KUKA KRL program: ab_com_01_st01_g01.src, ab_com_01_st01_g01.dat

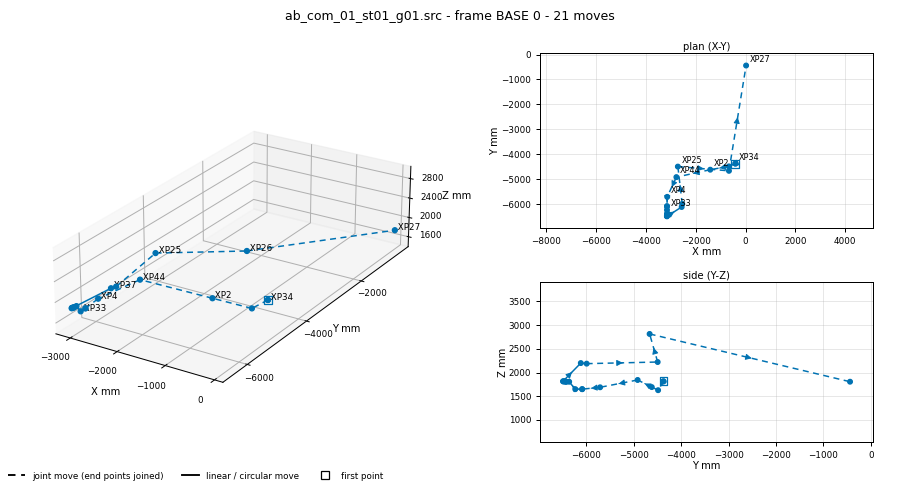
[picture p0: tool path of ab_com_01_st01_g01.src in frame BASE 0, 21 of 21 moves have a stored position in this frame; points joined in program order, loops and branches not executed]
--- ab_com_01_st01_g01.src ---
&ACCESS RVP1
&REL 2213
&COMMENT Deposito Frente AXOR_ATEGO
&PARAM DISKPATH = KRC:\R1\Program\OLP
&PARAM TEMPLATE = C:\KRC\Roboter\Template\vorgabe
&PARAM EDITMASK = *
DEF AB_COM_01_ST01_G01( )
;FOLD INI
  ;FOLD BASISTECH INI
    GLOBAL INTERRUPT DECL 3 WHEN $STOPMESS==TRUE DO IR_STOPM ( )
    INTERRUPT ON 3
    BAS (#INITMOV,0 )
  ;ENDFOLD (BASISTECH INI)
;FOLD SPOTTECH INI
USERSPOT(#INIT)
;ENDFOLD (SPOTTECH INI)
;FOLD GRIPPERTECH INI
USER_GRP(0,DUMMY,DUMMY,GDEFAULT)
;ENDFOLD (GRIPPERTECH INI)
  ;FOLD USER INI
    ;Make your modifications here

  ;ENDFOLD (USER INI)
;ENDFOLD (INI)

; Caracterização dos meios de produção
; Changes: Deposita Frontal na GeoBox
; Modelos:Atego/Axor - ETB/LTA/LTB/STB
; Versão Atual:28/03/2016
; Name: P13.050-R4

chk_w6_wechs_ok ( )  ; CHECK GRIPPER AXOR/ATEGO

;FOLD PTP P34 CONT Vel=100 % PDAT16 Tool[7]:Gripper Geo G01 01 Base[0] CD;%{PE}%R 8.2.20,%MKUKATPBASIS,%CMOVE,%VPTP,%P 1:PTP, 2:P34, 3:C_DIS, 5:100, 7:PDAT16
$BWDSTART=FALSE
PDAT_ACT=PPDAT16
FDAT_ACT=FP34
BAS(#PTP_PARAMS,100)
PTP XP34 C_DIS
;ENDFOLD

;FOLD PTP P7 Vel=100 % PDAT6 Tool[7]:Gripper Geo G01 01 Base[0];%{PE}%R 8.2.20,%MKUKATPBASIS,%CMOVE,%VPTP,%P 1:PTP, 2:P7, 3:, 5:100, 7:PDAT6
$BWDSTART=FALSE
PDAT_ACT=PPDAT6
FDAT_ACT=FP7
BAS(#PTP_PARAMS,100)
PTP XP7
;ENDFOLD

;FOLD OUT 3372 'Lib. pré Dep. Axor/Atego' State=TRUE ;%{PE}%R 8.2.20,%MKUKATPBASIS,%COUT,%VOUTX,%P 2:3372, 3:Lib. pré Dep. Axor/Atego, 5:TRUE, 6:
$OUT[3372]=TRUE
;ENDFOLD
;FOLD WAIT FOR ( IN 3372 'Lib. pré Deposito Axor/Atego' );%{PE}%R 8.2.20,%MKUKATPBASIS,%CEXT_WAIT_FOR,%VEXT_WAIT_FOR,%P 2:, 4:, 5:$IN, 6:3372, 7:Lib. pré Deposito Axor/Atego, 9:
WAIT FOR  ( $IN[3372] )
;ENDFOLD
;FOLD OUT 3372 'Lib. pré Dep. Axor/Atego' State=FALSE ;%{PE}%R 8.2.20,%MKUKATPBASIS,%COUT,%VOUTX,%P 2:3372, 3:Lib. pré Dep. Axor/Atego, 5:FALSE, 6:
$OUT[3372]=FALSE
;ENDFOLD
;FOLD OUT 3348 'Fora area GEOBOX' State=FALSE ;%{PE}%R 8.2.20,%MKUKATPBASIS,%COUT,%VOUTX,%P 2:3348, 3:Fora area GEOBOX, 5:FALSE, 6:
$OUT[3348]=FALSE
;ENDFOLD
;FOLD OUT 3340 'Area_Clear_AGV' State=FALSE ;%{PE}%R 8.2.20,%MKUKATPBASIS,%COUT,%VOUTX,%P 2:3340, 3:Area_Clear_AGV, 5:FALSE, 6:
$OUT[3340]=FALSE
;ENDFOLD

;FOLD PTP P1 CONT Vel=100 % PDAT1 Tool[7]:Gripper Geo G01 01 Base[0] CD;%{PE}%R 8.2.20,%MKUKATPBASIS,%CMOVE,%VPTP,%P 1:PTP, 2:P1, 3:C_DIS, 5:100, 7:PDAT1
$BWDSTART=FALSE
PDAT_ACT=PPDAT1
FDAT_ACT=FP1
BAS(#PTP_PARAMS,100)
PTP XP1 C_DIS
;ENDFOLD
;FOLD PTP P2 CONT Vel=100 % PDAT2 Tool[7]:Gripper Geo G01 01 Base[0] CD;%{PE}%R 8.2.20,%MKUKATPBASIS,%CMOVE,%VPTP,%P 1:PTP, 2:P2, 3:C_DIS, 5:100, 7:PDAT2
$BWDSTART=FALSE
PDAT_ACT=PPDAT2
FDAT_ACT=FP2
BAS(#PTP_PARAMS,100)
PTP XP2 C_DIS
;ENDFOLD
;FOLD PTP P44 CONT Vel=100 % PDAT27 Tool[7]:Gripper Geo G01 01 Base[0];%{PE}%R 8.2.20,%MKUKATPBASIS,%CMOVE,%VPTP,%P 1:PTP, 2:P44, 3:C_DIS, 5:100, 7:PDAT27
$BWDSTART=FALSE
PDAT_ACT=PPDAT27
FDAT_ACT=FP44
BAS(#PTP_PARAMS,100)
PTP XP44 C_DIS
;ENDFOLD
;FOLD PTP P4 CONT Vel=100 % PDAT8 Tool[7]:Gripper Geo G01 01 Base[0] CD;%{PE}%R 8.2.20,%MKUKATPBASIS,%CMOVE,%VPTP,%P 1:PTP, 2:P4, 3:C_DIS, 5:100, 7:PDAT8
$BWDSTART=FALSE
PDAT_ACT=PPDAT8
FDAT_ACT=FP4
BAS(#PTP_PARAMS,100)
PTP XP4 C_DIS
;ENDFOLD

;FOLD ; ABRE GRAMPOS E VERIFICA;%{PE}%R 8.2.20,%MKUKATPBASIS,%CCOMMENT,%VNORMAL,%P 2:ABRE  GRAMPOS  E  VERIFICA
;ENDFOLD
;FOLD SET Z3.1/Z3.2 AXOR State= GDAT20;%{PE}%R 8.2.1,%MKUKATPGRP,%CGRP,%VGRP,%P 2:7, 4:1, 5:#NO, 6:GDAT20, 8:0, 10:0
H50(GRP,7,1,GGDAT20)
;ENDFOLD
chk_w6_grp3_opn ()

;FOLD OUT 3374 'Lib. Dep. Axor/Atego' State=TRUE ;%{PE}%R 8.2.20,%MKUKATPBASIS,%COUT,%VOUTX,%P 2:3374, 3:Lib. Dep. Axor/Atego, 5:TRUE, 6:
$OUT[3374]=TRUE
;ENDFOLD
;FOLD WAIT FOR ( IN 3374 'Lib. Deposito Axor/Atego' );%{PE}%R 8.2.20,%MKUKATPBASIS,%CEXT_WAIT_FOR,%VEXT_WAIT_FOR,%P 2:, 4:, 5:$IN, 6:3374, 7:Lib. Deposito Axor/Atego, 9:
WAIT FOR  ( $IN[3374] )
;ENDFOLD
;FOLD OUT 3374 'Lib. Dep. Axor/Atego' State=FALSE ;%{PE}%R 8.2.20,%MKUKATPBASIS,%COUT,%VOUTX,%P 2:3374, 3:Lib. Dep. Axor/Atego, 5:FALSE, 6:
$OUT[3374]=FALSE
;ENDFOLD

;FOLD PTP P9 Vel=100 % PDAT11 Tool[7]:Gripper Geo G01 01 Base[0];%{PE}%R 8.2.20,%MKUKATPBASIS,%CMOVE,%VPTP,%P 1:PTP, 2:P9, 3:, 5:100, 7:PDAT11
$BWDSTART=FALSE
PDAT_ACT=PPDAT11
FDAT_ACT=FP9
BAS(#PTP_PARAMS,100)
PTP XP9
;ENDFOLD
;FOLD LIN P32 CONT Vel=0.5 m/s CPDAT20 Tool[7]:Gripper Geo G01 01 Base[0] CD;%{PE}%R 8.2.20,%MKUKATPBASIS,%CMOVE,%VLIN,%P 1:LIN, 2:P32, 3:C_DIS C_DIS, 5:0.5, 7:CPDAT20
$BWDSTART=FALSE
LDAT_ACT=LCPDAT20
FDAT_ACT=FP32
BAS(#CP_PARAMS,0.5)
LIN XP32 C_DIS C_DIS
;ENDFOLD
;FOLD LIN P33 CONT Vel=0.5 m/s CPDAT21 Tool[7]:Gripper Geo G01 01 Base[0] CD;%{PE}%R 8.2.20,%MKUKATPBASIS,%CMOVE,%VLIN,%P 1:LIN, 2:P33, 3:C_DIS C_DIS, 5:0.5, 7:CPDAT21
$BWDSTART=FALSE
LDAT_ACT=LCPDAT21
FDAT_ACT=FP33
BAS(#CP_PARAMS,0.5)
LIN XP33 C_DIS C_DIS
;ENDFOLD
;FOLD LIN P10 CONT Vel=0.5 m/s CPDAT4 Tool[7]:Gripper Geo G01 01 Base[0] CD;%{PE}%R 8.2.20,%MKUKATPBASIS,%CMOVE,%VLIN,%P 1:LIN, 2:P10, 3:C_DIS C_DIS, 5:0.5, 7:CPDAT4
$BWDSTART=FALSE
LDAT_ACT=LCPDAT4
FDAT_ACT=FP10
BAS(#CP_PARAMS,0.5)
LIN XP10 C_DIS C_DIS
;ENDFOLD
;FOLD LIN P5 CONT Vel=0.5 m/s CPDAT8 Tool[7]:Gripper Geo G01 01 Base[0] CD;%{PE}%R 8.2.20,%MKUKATPBASIS,%CMOVE,%VLIN,%P 1:LIN, 2:P5, 3:C_DIS C_DIS, 5:0.5, 7:CPDAT8
$BWDSTART=FALSE
LDAT_ACT=LCPDAT8
FDAT_ACT=FP5
BAS(#CP_PARAMS,0.5)
LIN XP5 C_DIS C_DIS
;ENDFOLD
;FOLD LIN P36 CONT Vel=0.5 m/s CPDAT22 Tool[7]:Gripper Geo G01 01 Base[0] CD;%{PE}%R 8.2.20,%MKUKATPBASIS,%CMOVE,%VLIN,%P 1:LIN, 2:P36, 3:C_DIS C_DIS, 5:0.5, 7:CPDAT22
$BWDSTART=FALSE
LDAT_ACT=LCPDAT22
FDAT_ACT=FP36
BAS(#CP_PARAMS,0.5)
LIN XP36 C_DIS C_DIS
;ENDFOLD
;FOLD LIN P17 CONT Vel=0.5 m/s CPDAT12 Tool[7]:Gripper Geo G01 01 Base[0] CD;%{PE}%R 8.2.20,%MKUKATPBASIS,%CMOVE,%VLIN,%P 1:LIN, 2:P17, 3:C_DIS C_DIS, 5:0.5, 7:CPDAT12
$BWDSTART=FALSE
LDAT_ACT=LCPDAT12
FDAT_ACT=FP17
BAS(#CP_PARAMS,0.5)
LIN XP17 C_DIS C_DIS
;ENDFOLD
;FOLD LIN P18 CONT Vel=0.5 m/s CPDAT13 Tool[7]:Gripper Geo G01 01 Base[0] CD;%{PE}%R 8.2.20,%MKUKATPBASIS,%CMOVE,%VLIN,%P 1:LIN, 2:P18, 3:C_DIS C_DIS, 5:0.5, 7:CPDAT13
$BWDSTART=FALSE
LDAT_ACT=LCPDAT13
FDAT_ACT=FP18
BAS(#CP_PARAMS,0.5)
LIN XP18 C_DIS C_DIS
;ENDFOLD
;FOLD LIN P11 CONT Vel=0.5 m/s CPDAT10 Tool[7]:Gripper Geo G01 01 Base[0] CD;%{PE}%R 8.2.20,%MKUKATPBASIS,%CMOVE,%VLIN,%P 1:LIN, 2:P11, 3:C_DIS C_DIS, 5:0.5, 7:CPDAT10
$BWDSTART=FALSE
LDAT_ACT=LCPDAT10
FDAT_ACT=FP11
BAS(#CP_PARAMS,0.5)
TQM_FIFO_READ(TM4)
TRIGGER WHEN DISTANCE=0 DELAY=TQM_DLY() DO iTQM_TRIGGERID=4
TRIGGER WHEN DISTANCE=0 DELAY=TQM_DLY() DO TQM_START_MON(TM4) PRIO = -1
TRIGGER WHEN DISTANCE=1 DELAY=0 DO TQM_SWAP_VALUES(TM4) PRIO = -1
LIN XP11 C_DIS C_DIS
;ENDFOLD

IF (NOT(GHOST())) THEN
;FOLD ; Deposita Gripper na GeoBox AXOR/ATEGO NEW;%{PE}%R 8.2.20,%MKUKATPBASIS,%CCOMMENT,%VNORMAL,%P 2:Deposita  Gripper  na  GeoBox  AXOR/ATEGO  NEW
;ENDFOLD
;FOLD LIN P38 Vel=0.1 m/s CPDAT24 Tool[7]:Gripper Geo G01 01 Base[0];%{PE}%R 8.2.20,%MKUKATPBASIS,%CMOVE,%VLIN,%P 1:LIN, 2:P38, 3:, 5:0.1, 7:CPDAT24
$BWDSTART=FALSE
LDAT_ACT=LCPDAT24
FDAT_ACT=FP38
BAS(#CP_PARAMS,0.1)
LIN XP38
;ENDFOLD
ENDIF

IF (GHOST()) THEN
;FOLD ; POSICAO DEPOSITO GRIPPER GEOBOX GHOST_RUN;%{PE}%R 8.2.20,%MKUKATPBASIS,%CCOMMENT,%VNORMAL,%P 2:POSICAO DEPOSITO GRIPPER GEOBOX  GHOST_RUN
;ENDFOLD
;FOLD LIN P37 Vel=0.5 m/s CPDAT25 Tool[8]:TOOL_CHANGE Base[0];%{PE}%R 8.2.20,%MKUKATPBASIS,%CMOVE,%VLIN,%P 1:LIN, 2:P37, 3:, 5:0.5, 7:CPDAT25
$BWDSTART=FALSE
LDAT_ACT=LCPDAT25
FDAT_ACT=FP37
BAS(#CP_PARAMS,0.5)
LIN XP37
;ENDFOLD
ENDIF

;FOLD OUT 3375 'Lib. p/ sair s/ Gripper Axor/Atego' State=TRUE ;%{PE}%R 8.2.20,%MKUKATPBASIS,%COUT,%VOUTX,%P 2:3375, 3:Lib. p/ sair s/ Gripper Axor/Atego, 5:TRUE, 6:
$OUT[3375]=TRUE
;ENDFOLD
;FOLD WAIT FOR ( IN 3375 'Lib. p/ sair s/ Gripper Axor/Atego' );%{PE}%R 8.2.20,%MKUKATPBASIS,%CEXT_WAIT_FOR,%VEXT_WAIT_FOR,%P 2:, 4:, 5:$IN, 6:3375, 7:Lib. p/ sair s/ Gripper Axor/Atego, 9:
WAIT FOR  ( $IN[3375] )
;ENDFOLD
;FOLD OUT 3375 'Lib. p/ sair s/ Gripper Axor/Atego' State=FALSE ;%{PE}%R 8.2.20,%MKUKATPBASIS,%COUT,%VOUTX,%P 2:3375, 3:Lib. p/ sair s/ Gripper Axor/Atego, 5:FALSE, 6:
$OUT[3375]=FALSE
;ENDFOLD

;FOLD ; FECHA GRAMPOS E VERIFICA;%{PE}%R 8.2.20,%MKUKATPBASIS,%CCOMMENT,%VNORMAL,%P 2:FECHA  GRAMPOS  E  VERIFICA
;ENDFOLD
;FOLD SET Z3.1/Z3.2 AXOR State=CLO GDAT12;%{PE}%R 8.2.1,%MKUKATPGRP,%CGRP,%VGRP,%P 2:7, 4:2, 5:#NO, 6:GDAT12, 8:0, 10:0
H50(GRP,7,2,GGDAT12)
;ENDFOLD
chk_w6_grp3_clo ( )

;FOLD OUT 224 'Bloquear MPS' State=FALSE ;%{PE}%R 8.2.20,%MKUKATPBASIS,%COUT,%VOUTX,%P 2:224, 3:Bloquear MPS, 5:FALSE, 6:
$OUT[224]=FALSE
;ENDFOLD
;FOLD OUT 223 'Desbloquear MPS' State=TRUE ;%{PE}%R 8.2.20,%MKUKATPBASIS,%COUT,%VOUTX,%P 2:223, 3:Desbloquear MPS, 5:TRUE, 6:
$OUT[223]=TRUE
;ENDFOLD
;FOLD WAIT FOR ( IN 217 'MPS Destravado' );%{PE}%R 8.2.20,%MKUKATPBASIS,%CEXT_WAIT_FOR,%VEXT_WAIT_FOR,%P 2:, 4:, 5:$IN, 6:217, 7:MPS Destravado, 9:
WAIT FOR  ( $IN[217] )
;ENDFOLD
;FOLD WAIT FOR NOT ( IN 221 'MPS Travado' );%{PE}%R 8.2.20,%MKUKATPBASIS,%CEXT_WAIT_FOR,%VEXT_WAIT_FOR,%P 2:NOT, 4:, 5:$IN, 6:221, 7:MPS Travado, 9:
WAIT FOR  NOT ( $IN[221] )
;ENDFOLD
;FOLD IBUS OFF;%{PE}%R 8.2.20,%MKUKATPBASIS,%CIBUS,%VMAP,%P 2:#OFF, 3:1
$IBUS_OFF=$IBUS_ON
$IBUS_ON=0
;ENDFOLD
;FOLD WAIT Time=0.2 sec;%{PE}%R 8.2.20,%MKUKATPBASIS,%CWAIT,%VWAIT,%P 3:0.2
WAIT SEC 0.2
;ENDFOLD

;FOLD LIN P24 Vel=0.1 m/s CPDAT5 Tool[8]:TOOL_CHANGE Base[0];%{PE}%R 8.2.20,%MKUKATPBASIS,%CMOVE,%VLIN,%P 1:LIN, 2:P24, 3:, 5:0.1, 7:CPDAT5
$BWDSTART=FALSE
LDAT_ACT=LCPDAT5
FDAT_ACT=FP24
BAS(#CP_PARAMS,0.1)
LIN XP24
;ENDFOLD

;FOLD WAIT FOR NOT ( IN 219 'Posicao p/ Acoplamento OK' ) CONT;%{PE}%R 8.2.20,%MKUKATPBASIS,%CEXT_WAIT_FOR,%VEXT_WAIT_FOR,%P 2:NOT, 4:, 5:$IN, 6:219, 7:Posicao p/ Acoplamento OK, 9:CONTINUE
CONTINUE
WAIT FOR  NOT ( $IN[219] )
;ENDFOLD
;FOLD OUT 223 'Desbloquear MPS' State=FALSE CONT;%{PE}%R 8.2.20,%MKUKATPBASIS,%COUT,%VOUTX,%P 2:223, 3:Desbloquear MPS, 5:FALSE, 6:CONTINUE
CONTINUE
$OUT[223]=FALSE
;ENDFOLD

;FOLD PTP P25 CONT Vel=100 % PDAT19 Tool[7]:Gripper Geo G01 01 Base[0] CD;%{PE}%R 8.2.20,%MKUKATPBASIS,%CMOVE,%VPTP,%P 1:PTP, 2:P25, 3:C_DIS, 5:100, 7:PDAT19
$BWDSTART=FALSE
PDAT_ACT=PPDAT19
FDAT_ACT=FP25
BAS(#PTP_PARAMS,100)
PTP XP25 C_DIS
;ENDFOLD
;FOLD PTP P26 CONT Vel=100 % PDAT20 Tool[7]:Gripper Geo G01 01 Base[0] CD;%{PE}%R 8.2.20,%MKUKATPBASIS,%CMOVE,%VPTP,%P 1:PTP, 2:P26, 3:C_DIS, 5:100, 7:PDAT20
$BWDSTART=FALSE
PDAT_ACT=PPDAT20
FDAT_ACT=FP26
BAS(#PTP_PARAMS,100)
PTP XP26 C_DIS
;ENDFOLD

;FOLD PULSE 199 'DOCK 5 Abrir Proteção' State=TRUE CONT Time=1 sec;%{PE}%R 8.2.20,%MKUKATPBASIS,%COUT,%VPULSE,%P 2:199, 3:DOCK 5 Abrir Proteção, 5:TRUE, 6:CONTINUE, 8:1
CONTINUE
PULSE($OUT[199], TRUE,1)
;ENDFOLD

;FOLD PTP P27 CONT Vel=100 % PDAT21 Tool[7]:Gripper Geo G01 01 Base[0] CD;%{PE}%R 8.2.20,%MKUKATPBASIS,%CMOVE,%VPTP,%P 1:PTP, 2:P27, 3:C_DIS, 5:100, 7:PDAT21
$BWDSTART=FALSE
PDAT_ACT=PPDAT21
FDAT_ACT=FP27
BAS(#PTP_PARAMS,100)
PTP XP27 C_DIS
;ENDFOLD

;FOLD PULSE 3343 'R4 entregou peca Geo' State=TRUE Time=3 sec;%{PE}%R 8.2.20,%MKUKATPBASIS,%COUT,%VPULSE,%P 2:3343, 3:R4 entregou peca Geo, 5:TRUE, 6:, 8:3
PULSE($OUT[3343], TRUE,3)
;ENDFOLD
;FOLD OUT 3348 'Fora area GEOBOX' State=TRUE ;%{PE}%R 8.2.20,%MKUKATPBASIS,%COUT,%VOUTX,%P 2:3348, 3:Fora area GEOBOX, 5:TRUE, 6:
$OUT[3348]=TRUE
;ENDFOLD

END

--- ab_com_01_st01_g01.dat ---
&ACCESS RVP1
&REL 2213
&COMMENT Deposito Frente AXOR_ATEGO
&PARAM DISKPATH = KRC:\R1\Program\OLP
&PARAM TEMPLATE = C:\KRC\Roboter\Template\vorgabe
&PARAM EDITMASK = *
DEFDAT  ab_com_01_st01_g01
;FOLD EXTERNAL DECLARATIONS;%{PE}%MKUKATPBASIS,%CEXT,%VCOMMON,%P
;FOLD GRIPPERTECH EXT
EXT  H50 (INT  :IN,INT  :IN,INT  :IN,GRP_TYP  :IN )
;ENDFOLD (GRIPPERTECH EXT)
;FOLD SPOTTECH EXT
EXT  USERSPOT (S_COMMAND  :IN,SPOT_TYPE  :IN )
;ENDFOLD (SPOTTECH EXT)
;FOLD BASISTECH EXT;%{PE}%MKUKATPBASIS,%CEXT,%VEXT,%P
EXT  BAS (BAS_COMMAND  :IN,REAL  :IN )
DECL INT SUCCESS
;ENDFOLD (BASISTECH EXT)
;FOLD USER EXT;%{E}%MKUKATPUSER,%CEXT,%VEXT,%P
;Make your modifications here

;ENDFOLD (USER EXT)
;ENDFOLD (EXTERNAL DECLARATIONS)
DECL BASIS_SUGG_T LAST_BASIS={POINT1[] "P44                     ",POINT2[] "P44                     ",CP_PARAMS[] "CPDAT24                 ",PTP_PARAMS[] "PDAT27                  ",CONT[] "                        ",CP_VEL[] "0.5                     ",PTP_VEL[] "100                     ",SYNC_PARAMS[] "SYNCDAT                 ",SPL_NAME[] "S0                      "}
DECL PDAT PPDAT1={VEL 100.0,ACC 100.0,APO_DIST 100.0,APO_MODE #CDIS}
DECL E6POS XP1={X -674.923401,Y -4487.53906,Z 1627.74695,A -32.1726799,B 80.8896866,C 37.8386002,S 2,T 34,E1 2143.02808,E2 0.0,E3 0.0,E4 0.0,E5 0.0,E6 0.0}
DECL FDAT FP1={TOOL_NO 7,BASE_NO 0,IPO_FRAME #BASE,POINT2[] " ",TQ_STATE FALSE}
DECL PDAT PPDAT2={VEL 100.0,ACC 100.0,APO_DIST 100.0,APO_MODE #CDIS}
DECL E6POS XP2={X -1421.39197,Y -4621.17188,Z 1693.43005,A -101.624001,B 83.8418121,C -18.5705299,S 2,T 34,E1 2975.92896,E2 0.0,E3 0.0,E4 0.0,E5 0.0,E6 0.0}
DECL FDAT FP2={TOOL_NO 7,BASE_NO 0,IPO_FRAME #BASE,POINT2[] " ",TQ_STATE FALSE}
DECL E6POS XP4={X -3149.48901,Y -5710.91699,Z 1688.84094,A 109.7183,B 88.3078537,C -159.620697,S 2,T 34,E1 4066.36694,E2 0.0,E3 0.0,E4 0.0,E5 0.0,E6 0.0}
DECL FDAT FP4={TOOL_NO 7,BASE_NO 0,IPO_FRAME #BASE,POINT2[] " ",TQ_STATE FALSE}
DECL E6POS XP5={X -3157.50391,Y -6424.60205,Z 1804.41699,A 108.200302,B 87.4537735,C -161.439697,S 2,T 34,E1 4703.12012,E2 0.0,E3 0.0,E4 0.0,E5 0.0,E6 0.0}
DECL FDAT FP5={TOOL_NO 7,BASE_NO 0,IPO_FRAME #BASE,POINT2[] " ",TQ_STATE FALSE}
DECL PDAT PPDAT6={VEL 100.0,ACC 100.0,APO_DIST 100.0,APO_MODE #CDIS}
DECL E6POS XP7={X -411.517609,Y -4374.29785,Z 1814.03601,A -89.7698822,B 87.6975327,C -41.859581,S 2,T 34,E1 2400.13794,E2 0.0,E3 0.0,E4 0.0,E5 0.0,E6 0.0}
DECL FDAT FP7={TOOL_NO 7,BASE_NO 0,IPO_FRAME #BASE,POINT2[] " ",TQ_STATE FALSE}
DECL GRP_SUGG_T LAST_GRP={NUMBER[] "7                       ",STATE[] "1                       ",PARAMS[] "GDAT12                  "}
DECL GRP_TYP GGDAT4={G_APO #NO,GRP_TIME 0.200000003,CTRL #OFF,DLY 0,DST 1}
DECL GRP_TYP GGDAT5={G_APO #NO,GRP_TIME 0.200000003,CTRL #OFF,DLY 0,DST 1}
DECL GRP_TYP GGDAT6={G_APO #NO,GRP_TIME 0.200000003,CTRL #OFF,DLY 0,DST 1}
DECL GRP_TYP GGDAT7={G_APO #NO,GRP_TIME 0.200000003,CTRL #OFF,DLY 0,DST 1}
DECL GRP_TYP GGDAT8={G_APO #NO,GRP_TIME 0.200000003,CTRL #OFF,DLY 0,DST 1}
DECL GRP_TYP GGDAT1={G_APO #NO,GRP_TIME 0.200000003,CTRL #OFF,DLY 0,DST 1}
DECL GRP_TYP GGDAT2={G_APO #NO,GRP_TIME 0.200000003,CTRL #OFF,DLY 0,DST 1}
DECL GRP_TYP GGDAT3={G_APO #NO,GRP_TIME 0.200000003,CTRL #OFF,DLY 0,DST 1}
DECL GRP_TYP GGDAT9={G_APO #NO,GRP_TIME 0.200000003,CTRL #OFF,DLY 0,DST 1}
DECL LDAT LCPDAT5={VEL 2.0,ACC 100.0,APO_DIST 100.0,APO_FAC 50.0,AXIS_VEL 100.0,AXIS_ACC 100.0,ORI_TYP #VAR,CIRC_TYP #BASE,JERK_FAC 50.0,GEAR_JERK 50.0,EXAX_IGN 0}
DECL E6POS XP24={X -2546.80005,Y -5994.47021,Z 2187.58398,A -178.397903,B 89.6208572,C -78.1456909,S 2,T 34,E1 4703.08984,E2 0.0,E3 0.0,E4 0.0,E5 0.0,E6 0.0}
DECL FDAT FP24={TOOL_NO 8,BASE_NO 0,IPO_FRAME #BASE,POINT2[] " ",TQ_STATE FALSE}
DECL PDAT PPDAT19={VEL 100.0,ACC 100.0,APO_DIST 100.0,APO_MODE #CDIS}
DECL E6POS XP25={X -2722.34497,Y -4496.51123,Z 2221.91895,A -156.239594,B 82.4170074,C -36.0250206,S 2,T 34,E1 3843.77905,E2 0.0,E3 0.0,E4 0.0,E5 0.0,E6 0.0}
DECL FDAT FP25={TOOL_NO 8,BASE_NO 0,IPO_FRAME #BASE,POINT2[] " ",TQ_STATE FALSE}
DECL PDAT PPDAT20={VEL 100.0,ACC 100.0,APO_DIST 100.0,APO_MODE #CDIS}
DECL E6POS XP26={X -670.858276,Y -4666.49707,Z 2814.13403,A -1.04210603,B -68.0760269,C 69.386467,S 6,T 18,E1 3241.76904,E2 0.0,E3 0.0,E4 0.0,E5 0.0,E6 0.0}
DECL FDAT FP26={TOOL_NO 8,BASE_NO 0,IPO_FRAME #BASE,POINT2[] " ",TQ_STATE FALSE}
DECL PDAT PPDAT21={VEL 100.0,ACC 100.0,APO_DIST 100.0,APO_MODE #CDIS}
DECL E6POS XP27={X 17.2738209,Y -439.133087,Z 1806.55896,A -150.870804,B -3.61021805,C -173.452301,S 2,T 2,E1 -343.7836,E2 0.0,E3 0.0,E4 0.0,E5 0.0,E6 0.0}
DECL FDAT FP27={TOOL_NO 8,BASE_NO 0,IPO_FRAME #BASE,POINT2[] " ",TQ_STATE FALSE}
DECL GRP_TYP GGDAT10={G_APO #NO,GRP_TIME 0.200000003,CTRL #OFF,DLY 0,DST 1}
DECL GRP_TYP GGDAT11={G_APO #NO,GRP_TIME 0.200000003,CTRL #OFF,DLY 0,DST 1}
DECL GRP_TYP GGDAT12={G_APO #NO,GRP_TIME 0.200000003,CTRL #OFF,DLY 0,DST 1}
DECL GRP_TYP GGDAT13={G_APO #NO,GRP_TIME 0.200000003,CTRL #OFF,DLY 0,DST 1}
DECL GRP_TYP GGDAT14={G_APO #NO,GRP_TIME 0.200000003,CTRL #OFF,DLY 0,DST 1}
DECL GRP_TYP GCONT={G_APO #YES,GRP_TIME 0.0,CTRL #OFF,DLY 0,DST 0}
DECL GRP_TYP GGDAT15={G_APO #NO,GRP_TIME 0.200000003,CTRL #OFF,DLY 0,DST 1}
DECL GRP_TYP GGDAT16={G_APO #NO,GRP_TIME 0.200000003,CTRL #OFF,DLY 0,DST 1}
DECL E6POS XP30={X -2781.42603,Y -4919.25293,Z 1843.13403,A -95.6107864,B 80.072052,C -9.8578167,S 2,T 34,E1 3587.7981,E2 0.0,E3 0.0,E4 0.0,E5 0.0,E6 0.0}
DECL FDAT FP30={TOOL_NO 7,BASE_NO 0,IPO_FRAME #BASE,POINT2[] " ",TQ_STATE TRUE}
DECL LDAT LCPDAT8={VEL 2.0,ACC 50.0,APO_DIST 50.0,APO_FAC 50.0,AXIS_VEL 100.0,AXIS_ACC 100.0,ORI_TYP #VAR,CIRC_TYP #BASE,JERK_FAC 50.0,GEAR_JERK 50.0,EXAX_IGN 0}
DECL PDAT PPDAT7={VEL 100.0,ACC 100.0,APO_DIST 100.0,APO_MODE #CDIS}
DECL PDAT PPDAT8={VEL 100.0,ACC 80.0,APO_DIST 30.0,APO_MODE #CDIS}
DECL E6POS XP9={X -3158.62598,Y -6089.2168,Z 1649.49902,A 95.3501282,B 87.6326523,C -174.400406,S 2,T 34,E1 4703.12598,E2 0.0,E3 0.0,E4 0.0,E5 0.0,E6 0.0}
DECL FDAT FP9={TOOL_NO 7,BASE_NO 0,IPO_FRAME #BASE,POINT2[] " ",TQ_STATE FALSE}
DECL PDAT PPDAT11={VEL 100.0,ACC 100.0,APO_DIST 100.0}
DECL E6POS XP10={X -3151.78394,Y -6363.49316,Z 1805.849,A 111.823402,B 87.3075714,C -157.943298,S 2,T 34,E1 4703.12402,E2 0.0,E3 0.0,E4 0.0,E5 0.0,E6 0.0}
DECL FDAT FP10={TOOL_NO 7,BASE_NO 0,IPO_FRAME #BASE,POINT2[] " ",TQ_STATE FALSE}
DECL LDAT LCPDAT4={VEL 2.0,ACC 50.0,APO_DIST 50.0,APO_FAC 50.0,AXIS_VEL 100.0,AXIS_ACC 100.0,ORI_TYP #VAR,CIRC_TYP #BASE,JERK_FAC 50.0,GEAR_JERK 50.0,EXAX_IGN 0}
DECL TQM_TQDAT_T TM3={T11 200,T12 200,T13 200,T14 200,T15 200,T16 200,T21 114497,T22 114497,T23 114497,T24 114497,T25 114497,T26 114497,K1 319,K2 313,K3 315,K4 315,K5 314,K6 316,O1 20,O2 30,ID 3,OVM 0,TMF 75976.0}
DECL E6POS XP11={X -3162.25806,Y -6479.81299,Z 1813.18506,A 128.677505,B 89.5311279,C -141.025299,S 2,T 34,E1 4703.104,E2 0.0,E3 0.0,E4 0.0,E5 0.0,E6 0.0}
DECL FDAT FP11={TOOL_NO 7,BASE_NO 0,IPO_FRAME #BASE,POINT2[] " ",TQ_STATE TRUE}
DECL LDAT LCPDAT10={VEL 2.0,ACC 50.0,APO_DIST 50.0,APO_FAC 50.0,AXIS_VEL 100.0,AXIS_ACC 100.0,ORI_TYP #VAR,CIRC_TYP #BASE,JERK_FAC 50.0,GEAR_JERK 50.0,EXAX_IGN 0}
DECL TQM_TQDAT_T TM4={T11 9,T12 4,T13 3,T14 3,T15 6,T16 2,T21 1,T22 1,T23 0,T24 0,T25 0,T26 0,K1 301,K2 299,K3 300,K4 300,K5 300,K6 299,O1 20,O2 30,ID 4,OVM 100,TMF 1.5}
DECL GRP_TYP GGDAT17={G_APO #NO,GRP_TIME 0.200000003,CTRL #OFF,DLY 0,DST 1}
DECL GRP_TYP GGDAT18={G_APO #NO,GRP_TIME 0.200000003,CTRL #OFF,DLY 0,DST 1}
DECL GRP_TYP GGDAT19={G_APO #NO,GRP_TIME 0.200000003,CTRL #OFF,DLY 0,DST 1}
DECL E6POS XP17={X -3159.59204,Y -6448.65381,Z 1811.28894,A 119.683998,B 88.6462021,C -149.935593,S 2,T 34,E1 4703.125,E2 0.0,E3 0.0,E4 0.0,E5 0.0,E6 0.0}
DECL FDAT FP17={TOOL_NO 7,BASE_NO 0,IPO_FRAME #BASE,POINT2[] " ",TQ_STATE FALSE}
DECL LDAT LCPDAT12={VEL 2.0,ACC 100.0,APO_DIST 50.0,APO_FAC 50.0,AXIS_VEL 100.0,AXIS_ACC 100.0,ORI_TYP #VAR,CIRC_TYP #BASE,JERK_FAC 50.0,GEAR_JERK 50.0,EXAX_IGN 0}
DECL E6POS XP18={X -3162.25391,Y -6479.81494,Z 1814.72205,A 128.658005,B 89.5313721,C -141.044907,S 2,T 34,E1 4703.104,E2 0.0,E3 0.0,E4 0.0,E5 0.0,E6 0.0}
DECL FDAT FP18={TOOL_NO 7,BASE_NO 0,IPO_FRAME #BASE,POINT2[] " ",TQ_STATE FALSE}
DECL LDAT LCPDAT13={VEL 2.0,ACC 100.0,APO_DIST 50.0,APO_FAC 50.0,AXIS_VEL 100.0,AXIS_ACC 100.0,ORI_TYP #VAR,CIRC_TYP #BASE,JERK_FAC 50.0,GEAR_JERK 50.0,EXAX_IGN 0}
DECL LDAT LCPDAT20={VEL 2.0,ACC 100.0,APO_DIST 50.0,APO_FAC 50.0,AXIS_VEL 100.0,AXIS_ACC 100.0,ORI_TYP #VAR,CIRC_TYP #BASE,JERK_FAC 50.0,GEAR_JERK 50.0,EXAX_IGN 0}
DECL E6POS XP32={X -3158.61499,Y -6089.20996,Z 1649.46106,A 95.3123474,B 87.6316681,C -174.438904,S 2,T 34,E1 4703.125,E2 0.0,E3 0.0,E4 0.0,E5 0.0,E6 0.0}
DECL FDAT FP32={TOOL_NO 7,BASE_NO 0,IPO_FRAME #BASE,POINT2[] " ",TQ_STATE FALSE}
DECL LDAT LCPDAT21={VEL 2.0,ACC 100.0,APO_DIST 50.0,APO_FAC 50.0,AXIS_VEL 100.0,AXIS_ACC 100.0,ORI_TYP #VAR,CIRC_TYP #BASE,JERK_FAC 50.0,GEAR_JERK 50.0,EXAX_IGN 0}
DECL E6POS XP33={X -3158.62988,Y -6234.4668,Z 1649.48499,A 95.3606186,B 87.6313019,C -174.390594,S 2,T 34,E1 4703.125,E2 0.0,E3 0.0,E4 0.0,E5 0.0,E6 0.0}
DECL FDAT FP33={TOOL_NO 7,BASE_NO 0,IPO_FRAME #BASE,POINT2[] " ",TQ_STATE FALSE}
DECL E6POS XP34={X -411.520813,Y -4374.2998,Z 1814.03796,A -89.7720032,B 87.6974106,C -41.8615189,S 2,T 34,E1 2400.13794,E2 0.0,E3 0.0,E4 0.0,E5 0.0,E6 0.0}
DECL FDAT FP34={TOOL_NO 7,BASE_NO 0,IPO_FRAME #BASE,POINT2[] " ",TQ_STATE FALSE}
DECL PDAT PPDAT16={VEL 100.0,ACC 100.0,APO_DIST 100.0,APO_MODE #CDIS}
DECL LDAT LCPDAT22={VEL 2.0,ACC 50.0,APO_DIST 50.0,APO_FAC 50.0,AXIS_VEL 100.0,AXIS_ACC 100.0,ORI_TYP #VAR,CIRC_TYP #BASE,JERK_FAC 50.0,GEAR_JERK 50.0,EXAX_IGN 0}
DECL E6POS XP36={X -3155.67212,Y -6434.43408,Z 1808.93604,A 111.804802,B 88.0430527,C -157.778702,S 2,T 34,E1 4703.12402,E2 0.0,E3 0.0,E4 0.0,E5 0.0,E6 0.0}
DECL FDAT FP36={TOOL_NO 7,BASE_NO 0,IPO_FRAME #BASE,POINT2[] " ",TQ_STATE FALSE}
DECL E6POS XP37={X -2569.37793,Y -6118.03906,Z 2199.79199,A 171.807602,B 89.9708328,C -87.9462204,S 2,T 34,E1 4696.35205,E2 0.0,E3 0.0,E4 0.0,E5 0.0,E6 0.0}
DECL FDAT FP37={TOOL_NO 8,BASE_NO 0,IPO_FRAME #BASE,POINT2[] " ",TQ_STATE FALSE}
DECL LDAT LCPDAT23={VEL 2.0,ACC 100.0,APO_DIST 100.0,APO_FAC 50.0,AXIS_VEL 100.0,AXIS_ACC 100.0,ORI_TYP #VAR,CIRC_TYP #BASE,JERK_FAC 50.0,GEAR_JERK 50.0,EXAX_IGN 0}
DECL LDAT LCPDAT24={VEL 2.0,ACC 100.0,APO_DIST 100.0,APO_FAC 50.0,AXIS_VEL 100.0,AXIS_ACC 100.0,ORI_TYP #VAR,CIRC_TYP #BASE,JERK_FAC 50.0,GEAR_JERK 50.0,EXAX_IGN 0}
DECL E6POS XP38={X -3160.27197,Y -6494.2002,Z 1815.09399,A 178.284698,B 89.8384705,C -91.4645386,S 2,T 34,E1 4703.11084,E2 0.0,E3 0.0,E4 0.0,E5 0.0,E6 0.0}
DECL FDAT FP38={TOOL_NO 7,BASE_NO 0,IPO_FRAME #BASE,POINT2[] " ",TQ_STATE FALSE}
DECL PDAT PPDAT18={VEL 100.0,ACC 100.0,APO_DIST 100.0}
DECL LDAT LCPDAT25={VEL 2.0,ACC 100.0,APO_DIST 100.0,APO_FAC 50.0,AXIS_VEL 100.0,AXIS_ACC 100.0,ORI_TYP #VAR,CIRC_TYP #BASE,JERK_FAC 50.0,GEAR_JERK 50.0,EXAX_IGN 0}
DECL E6POS XP39={X -2571.16504,Y -6117.65723,Z 2190.50391,A 67.8934631,B 89.7762604,C 168.294205,S 2,T 10,E1 4703.13184,E2 0.0,E3 0.0,E4 0.0,E5 0.0,E6 0.0}
DECL FDAT FP39={TOOL_NO 8,BASE_NO 0,IPO_FRAME #BASE,POINT2[] " ",TQ_STATE FALSE}
DECL PDAT PPDAT22={VEL 100.0,ACC 100.0,APO_DIST 100.0}
DECL E6POS XP40={X -2571.0979,Y -6117.65723,Z 2190.83911,A 68.1121674,B 89.7844086,C 168.507004,S 2,T 10,E1 4702.87207,E2 0.0,E3 0.0,E4 0.0,E5 0.0,E6 0.0}
DECL FDAT FP40={TOOL_NO 8,BASE_NO 0,IPO_FRAME #BASE,POINT2[] " ",TQ_STATE FALSE}
DECL PDAT PPDAT23={VEL 100.0,ACC 100.0,APO_DIST 100.0}
DECL E6POS XP41={X -2571.21997,Y -6117.67822,Z 2190.13696,A 66.7464981,B 89.7574234,C 167.147797,S 2,T 10,E1 4703.13086,E2 0.0,E3 0.0,E4 0.0,E5 0.0,E6 0.0}
DECL FDAT FP41={TOOL_NO 8,BASE_NO 0,IPO_FRAME #BASE,POINT2[] " ",TQ_STATE FALSE}
DECL PDAT PPDAT24={VEL 100.0,ACC 100.0,APO_DIST 100.0}
DECL E6POS XP42={X -1766.05103,Y -4545.29688,Z 2302.94092,A -126.665298,B 6.63578176,C 123.795197,S 2,T 34,E1 3703.29102,E2 0.0,E3 0.0,E4 0.0,E5 0.0,E6 0.0}
DECL FDAT FP42={TOOL_NO 8,BASE_NO 0,IPO_FRAME #BASE,POINT2[] " ",TQ_STATE FALSE}
DECL PDAT PPDAT25={VEL 100.0,ACC 100.0,APO_DIST 100.0}
DECL E6POS XP43={X -3160.26392,Y -6494.22412,Z 1815.14905,A 178.839096,B 89.8379364,C -90.9104538,S 2,T 34,E1 4703.12109,E2 0.0,E3 0.0,E4 0.0,E5 0.0,E6 0.0}
DECL FDAT FP43={TOOL_NO 7,BASE_NO 0,IPO_FRAME #BASE,POINT2[] " ",TQ_STATE FALSE}
DECL PDAT PPDAT26={VEL 100.0,ACC 100.0,APO_DIST 100.0}
DECL E6POS XP44={X -2781.4231,Y -4919.25488,Z 1843.13098,A -95.6104736,B 80.0721893,C -9.857687,S 2,T 34,E1 3587.7981,E2 0.0,E3 0.0,E4 0.0,E5 0.0,E6 0.0}
DECL FDAT FP44={TOOL_NO 7,BASE_NO 0,IPO_FRAME #BASE,POINT2[] " ",TQ_STATE FALSE}
DECL PDAT PPDAT27={VEL 100.0,ACC 100.0,APO_DIST 100.0,APO_MODE #CDIS}
DECL GRP_TYP GGDAT20={G_APO #NO,GRP_TIME 0.200000003,CTRL #OFF,DLY 0,DST 1}
ENDDAT
